PROGRAM MAIN
VAR
    fb_CallHandler : CallHandler;
    fb_MovementControl : MovementControl;
    fb_DoorControl : DoorControl;
	fb_DoorSensors : DoorSensors;
	fb_Lights : Lights;
	fb_TargetFloorLights : TargetFloorLights;
END_VAR

fb_CallHandler();
fb_DoorControl();
fb_MovementControl();
fb_DoorSensors();
fb_Lights();
fb_TargetFloorLights();

END_PROGRAM

(* stored: Version 1.1.0.1, ProductVersion 3.1.4024.15
   POU MAIN: Id {cdb5c23c-b562-4f2f-82d6-ee339a1fb725}, SpecialFunc None *)
